{attribute 'linkalways'} 
{attribute 'no_explicit_call' := 'This FB is a CLASS and must be accessed using methods or properties'}
{attribute 'enable_dynamic_creation'}
FUNCTION_BLOCK MockNumericDatatype_INT EXTENDS NumericDatatypeBase
VAR
	localData : INT;
	activeData : REFERENCE TO INT REF= localData;
END_VAR

PROPERTY PUBLIC Address : PVOID
GET
Address := ADR(activeData);
END_GET
END_PROPERTY

METHOD PUBLIC ClearReference
VAR_INPUT
END_VAR
activeData REF= localData;
END_METHOD

METHOD PUBLIC Clone : I_Datatype
VAR
    pClone : POINTER TO MockNumericDatatype_INT;
END_VAR
pClone := __NEW(MockNumericDatatype_INT(InitialValue := Value));
Clone := pClone^;
END_METHOD

METHOD FB_init : BOOL
VAR_INPUT
	bInitRetains : BOOL; // if TRUE, the retain variables are initialized (warm start / cold start)
	bInCopyCode : BOOL;  // if TRUE, the instance afterwards gets moved into the copy code (online change)
	InitialValue : INT;
END_VAR
localData := InitialValue;
END_METHOD

PROPERTY PUBLIC IsFloat : BOOL
GET
IsFloat := FALSE;
END_GET
END_PROPERTY

PROPERTY PUBLIC IsSigned : BOOL
GET
IsSigned := TRUE;
END_GET
END_PROPERTY

METHOD PUBLIC MakeReferenceTo
VAR_INPUT
	ReferenceTarget : REFERENCE TO INT;
END_VAR
activeData REF= ReferenceTarget;
END_METHOD

PROPERTY PUBLIC MaxValue : INT
GET
MaxValue := DatatypeLimits.INT_MAX_VALUE;
END_GET
END_PROPERTY

PROPERTY PUBLIC MinValue : INT
GET
MinValue := DatatypeLimits.INT_MIN_VALUE;
END_GET
END_PROPERTY

METHOD PROTECTED SerializeMaxValue
VAR_INPUT
	Serializer : I_Serializer;
END_VAR
Serializer.AddInt(MaxValue);
END_METHOD

METHOD PROTECTED SerializeMinValue
VAR_INPUT
	Serializer : I_Serializer;
END_VAR
Serializer.AddInt(MinValue);
END_METHOD

METHOD PUBLIC SerializeWith
VAR_INPUT
	Serializer : I_Serializer;
END_VAR
Serializer.AddInt(activeData);
END_METHOD

PROPERTY PUBLIC Size : UDINT
GET
Size := SIZEOF(activeData);
END_GET
END_PROPERTY

METHOD TryDeserializeFrom : BOOL
VAR_INPUT
	Deserializer : I_Deserializer;
	Feedback : I_DeserializerFeedback;
END_VAR
TryDeserializeFrom := Deserializer.TryGetInt(activeData, Feedback);
END_METHOD

METHOD TryMakeReferenceTo : BOOL
VAR_INPUT
	Target : I_Datatype;
END_VAR
VAR
	pTargetData : POINTER TO INT;
END_VAR
IF NOT (Target.TypeName = TypeName) THEN
	RETURN;
END_IF

pTargetData := Target.Address;
activeData REF= pTargetData^;
TryMakeReferenceTo := TRUE;
END_METHOD

PROPERTY PUBLIC TypeName : T_MAXSTRING
GET
TypeName := 'INT';
END_GET
END_PROPERTY

PROPERTY PUBLIC Value : INT
GET
Value := activeData;
END_GET
SET
activeData := Value;
END_SET
END_PROPERTY

END_FUNCTION_BLOCK

(* stored: Version 1.1.0.1, ProductVersion 3.1.4024.12
   POU MockNumericDatatype_INT: Id {2c662a08-c485-49a1-b995-016487ecc69b}, SpecialFunc None
   Folder Constructor: Id {be11e387-00ef-4f93-b95b-121a57200523}
   Folder Protected: Id {e042c7f8-464d-4a88-b806-1c57492ab18f}
   Property Address: Id {2ed59742-f7d1-4ca3-b1c1-4f0f616672f5}
   Get Get: Id {4006c0ef-9e60-4507-b5a9-d0ed65019c80}
   Method ClearReference: Id {a9a2765a-f793-43f5-9524-9a2866ebaab8}
   Method Clone: Id {f01b83a8-b22c-41c2-9d04-a66308b1f451}
   Method FB_init: Id {cc2dd1fa-b428-44e7-a3c6-4ae91280b50f}
   Property IsFloat: Id {ebe80431-ce31-42ae-b310-096ca3adcdc2}
   Get Get: Id {d0cf8171-8a01-4d2c-9a05-da10ae0a3dd3}
   Property IsSigned: Id {be8bfbb0-ede8-4a49-b794-48cecb2f9a06}
   Get Get: Id {e56a8c72-1bab-48d2-a125-ea23714c7b8d}
   Method MakeReferenceTo: Id {e19f5cfe-69c3-4cc7-a388-01d457167e83}
   Property MaxValue: Id {a54fbfa9-5d34-4154-bf82-6152a920c6b9}
   Get Get: Id {32afd05e-e11a-4c59-8826-47f57741936f}
   Property MinValue: Id {36f2f4ec-b0e7-42a3-a59d-71a21c00906d}
   Get Get: Id {5fa0df12-bf50-4016-b01d-109a28996cdb}
   Method SerializeMaxValue: Id {bfbbdc3b-0c7e-4c5e-9e4c-b4752537746e}
   Method SerializeMinValue: Id {fe532488-653c-4a08-bf6a-5bf20578c9df}
   Method SerializeWith: Id {55d859ad-14a8-4fcc-90a9-d4b8955ed62d}
   Property Size: Id {82607b90-3206-40db-a27f-ba335b7aa8de}
   Get Get: Id {d2b2f4a6-24e4-45f1-b18f-1979299436b6}
   Method TryDeserializeFrom: Id {030df632-6db4-45e9-ad02-5a6509a59fef}
   Method TryMakeReferenceTo: Id {a5de350a-77a8-41b6-a300-eb76f8fbfcc6}
   Property TypeName: Id {e77e83b7-13ae-482b-96f2-2e7af99fb611}
   Get Get: Id {dd3070f4-934f-4043-928f-35acfcf5a147}
   Property Value: Id {4bcf8094-2958-45b7-865a-81399da8c529}
   Get Get: Id {bf9ec9e1-15ef-4553-8235-ece87bb773d8}
   Set Set: Id {8e2beeb1-1c0c-40fd-bb15-6101cf4f43d3} *)
